INTERFACE ITF_StandardFB

METHOD EMstop : Bool
VAR_INPUT
END_VAR
END_METHOD

METHOD getDiagnostics
VAR_IN_OUT
	AddError		: ARRAY [*] OF FB_AddErrorST;
	a_ActiveEvents	: ARRAY [*] OF ST_ErrorStruct;
	w_Index			: WORD;
END_VAR
END_METHOD

METHOD Init : Bool
VAR_INPUT
END_VAR
END_METHOD

METHOD Reset : Bool
VAR_INPUT
END_VAR
END_METHOD

END_INTERFACE

(* stored: Version 1.1.0.1, ProductVersion 3.1.4026.18
   Itf ITF_StandardFB: Id {1ff54861-7e61-400a-a15a-c0cb5d445c6a}
   Method EMstop: Id {0ee59298-071d-415d-8b60-1fa427633d9b}
   Method getDiagnostics: Id {e8887f99-5c4f-4384-b52a-b164a9b15492}
   Method Init: Id {4d0bd109-c989-4c1a-9e98-b73d9a0fd00d}
   Method Reset: Id {bf1c81e8-9c87-4182-ad78-8df62fad367a} *)
